VISUALIZATION Conv_handling  // 884x633
END_VISUALIZATION

(* stored: Version 1.1.0.1, ProductVersion 3.1.4024.11
   Visu Conv_handling: Id {5300551a-10e5-47ae-9dd0-56e14f55f2f0} *)
